{attribute 'GeneratedUsingTerminal: ELX9560-0000-0016'}
{attribute addProperty BoxType "ELX9560-0000-0016"}
{attribute addProperty Id "Power_OKAT %I*BOOL1"}
{attribute addProperty CRC "1151167157"}
{attribute addProperty Size "1"}
TYPE Status_Uin_449D6AB5 :
STRUCT
	{attribute addProperty Name "Power_OK"}
	Power_OK AT %I* : BOOL;
END_STRUCT
END_TYPE

(* stored: Version 1.2.0.0, ProductVersion 3.1.4024.9
   DUT Status_Uin_449D6AB5: Id {930f9380-9b31-4d4f-b2cd-c59917249b80} *)
